FUNCTION_BLOCK CompositeTestBlock4
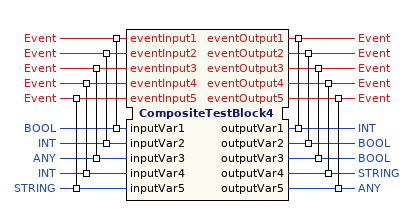
  EVENT_INPUT
    eventInput1 WITH inputVar1;
    eventInput2 WITH inputVar2;
    eventInput3 WITH inputVar3;
    eventInput4 WITH inputVar4;
    eventInput5 WITH inputVar5;
  END_EVENT
  EVENT_OUTPUT
    eventOutput1 WITH outputVar1;
    eventOutput2 WITH outputVar2;
    eventOutput3 WITH outputVar3;
    eventOutput4 WITH outputVar4;
    eventOutput5 WITH outputVar5;
  END_EVENT
  VAR_INPUT
    inputVar1 : BOOL;
    inputVar2 : INT;
    inputVar3 : ANY;
    inputVar4 : INT;
    inputVar5 : STRING;
  END_VAR
  VAR_OUTPUT
    outputVar1 : INT;
    outputVar2 : BOOL;
    outputVar3 : BOOL;
    outputVar4 : STRING;
    outputVar5 : ANY;
  END_VAR
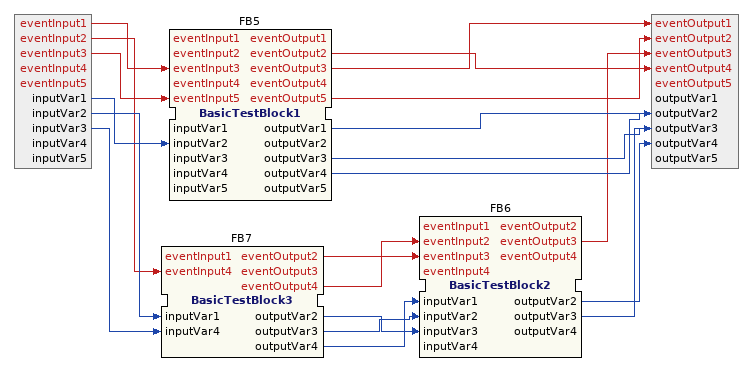
  FBS
    FB5 : BasicTestBlock1;
    FB6 : BasicTestBlock2;
    FB7 : BasicTestBlock3;
  END_FBS
  EVENT_CONNECTIONS
    FB7.eventOutput4 TO FB6.eventInput2;
    FB7.eventOutput2 TO FB6.eventInput3;
    eventInput3 TO FB5.eventInput5;
    eventInput1 TO FB5.eventInput3;
    eventInput2 TO FB7.eventInput4;
    FB5.eventOutput2 TO eventOutput4;
    FB5.eventOutput3 TO eventOutput1;
    FB5.eventOutput5 TO eventOutput2;
    FB6.eventOutput3 TO eventOutput3;
  END_CONNECTIONS
  DATA_CONNECTIONS
    FB7.outputVar2 TO FB6.inputVar3;
    FB7.outputVar3 TO FB6.inputVar2;
    FB7.outputVar4 TO FB6.inputVar1;
    inputVar1 TO FB5.inputVar2;
    FB6.outputVar2 TO outputVar4;
    FB6.outputVar3 TO outputVar3;
    FB5.outputVar1 TO outputVar2;
    FB5.outputVar4 TO outputVar2;
    FB5.outputVar3 TO outputVar3;
    inputVar3 TO FB7.inputVar4;
    inputVar2 TO FB7.inputVar1;
  END_CONNECTIONS
END_FUNCTION_BLOCK
